TYPE T_CodeCRYPTO : STRING[20];
END_TYPE

(* stored: Version 1.1.0.1
   DUT T_CodeCRYPTO: Id {5649ef93-04d1-4ad8-b961-441a6d2de0c6} *)
